(* CODESYS project fablev5.project
   CompiledLibraryCompatibilityVersion: LeadSysStudio V3.5 SP15 Patch 4
   Title: MC500_EtherCAT_axis_motion

Project tree, tasks and I/O mapping:
  Device : MC508, Leadshine Technology Co., Ltd., order no. 508101, version 3.5.15.40
      settings: RetainMode = 0; RetainStartAddr = 20480; RetainEndAddr = 524288; RetainSize = 524288
    application Application
      libraries: Standard, * (System); LS_ModbusMasterlib, 0.0.0.2 (Leadshine Technology Co.Ltd)
      task MainTask (cyclic, interval 4000 µs, priority 1) calls EtherCAT_Master_Leadshine_A.EtherCAT_Task, POU
      program PLC_PRG [LD]: EC_Axis_motion_control
      program POU [ST]
      program POU_1 [ST]
      program POU_3 [ST]
    Resource Usage
    Network Configuration
      LocalBus Config
    Device Diagnose
    LocalBus_Master_Module : LocalBus Master, Leadshine Technology Co., Ltd., version 3.5.15.40
    ModbusCOM_Master_1 : ModbusCOM RS-485 Master, Leadshine Technology Co., Ltd., version 3.5.15.40
        settings: com.Parity = 2; com.FrameIntervTime = 10; com.Baudrate = 115200
      ModbusCOM_Slave : ModbusCOM Slave, Leadshine Technology Co., Ltd., version 3.5.15.40
          settings: ModBusRTU_ErrorCode = 0; Z_Trigger.FuncCode = 6; Z_Trigger.ControlMode = 1; Z_Trigger.ResendCount = 1; Z_Trigger.WriteRegOffSet = 24578; Z_Trigger.IOChannel = 0; Z_Trigger.ChannelName = 'Z_Trigger'; Z_Trigger.ChannelNote = ''; Z_Status.FuncCode = 3; Z_Status.ResendCount = 1; Z_Status.CycleTimes = 50; Z_Status.ReadRegOffSet = 24578; Z_Status.ChannelName = 'Z_Status'; Z_Status.ChannelNote = ''; Z_MotionStat.FuncCode = 3; Z_MotionStat.ResendCount = 1; Z_MotionStat.CycleTimes = 50; Z_MotionStat.ReadRegOffSet = 4099; Z_MotionStat.IOChannel = 2; Z_MotionStat.ChannelName = 'Z_MotionStat'; Z_MotionStat.ChannelNote = ''; Z_Enable.FuncCode = 6; Z_Enable.ControlMode = 1; Z_Enable.ResendCount = 1; Z_Enable.WriteRegOffSet = 15; Z_Enable.IOChannel = 3; Z_Enable.ChannelName = 'Z_Enable'; Z_Enable.ChannelNote = ''; Z_DIStatus.FuncCode = 3; Z_DIStatus.ResendCount = 1; Z_DIStatus.CycleTimes = 200; Z_DIStatus.ReadRegOffSet = 377; Z_DIStatus.IOChannel = 4; Z_DIStatus.ChannelName = 'Z_DIStatus'; Z_DIStatus.ChannelNote = ''; Vendor.SlaveID = 2; Vendor.ChannelNum = 5; Vendor.Timeout = 100
          unmapped channels: ErrorCode, Z_Trigger, Z_Trigger, Z_Trigger, Z_Status, Z_Status, Z_MotionStat, Z_MotionStat, Z_Enable, Z_Enable, Z_Enable, Z_DIStatus, Z_DIStatus
    High_Speed_IO_Module : High Speed IO, Leadshine Technology Co., Ltd., version 3.5.15.40
        unmapped channels: Genral_IO_IN, Genral_IO_Out
    SoftMotion General Axis Pool
    EtherCAT_Master_Leadshine_A : EtherCAT Master SoftMotion, 3S - Smart Software Solutions GmbH, version 3.5.15.30
        settings: NetworkName = 'ecat'; SelectNetworkByName = TRUE
      CS3E_D1008 : CS3E-D1008(COE), Leadshine Technology Co.,Ltd., order no. CS3E-D1008, version Revision=16#00000001
          settings: DC sync0 cycletime = 4000; DC sync1 cycletime = 4000; Number of SDO = 6; Homing method.Index = 16#6098; Homing method.Subindex = 16#00; Homing method.Value = 17; Homing method.Size = 8; Homing method.AbortIfError = FALSE; Homing method.JumpToLine = FALSE; Homing method.Line = 0; Homing method.CompleteAccess = FALSE; Homing velocity (fast).Index = 16#6099; Homing velocity (fast).Subindex = 16#01; Homing velocity (fast).Value = 2000; Homing velocity (fast).Size = 32; Homing velocity (fast).AbortIfError = FALSE; Homing velocity (fast).JumpToLine = FALSE; Homing velocity (fast).Line = 0; Homing velocity (fast).CompleteAccess = FALSE; Homing velocity (slow).Index = 16#6099; Homing velocity (slow).Subindex = 16#02; Homing velocity (slow).Value = 300; Homing velocity (slow).Size = 32; Homing velocity (slow).AbortIfError = FALSE; Homing velocity (slow).JumpToLine = FALSE; Homing velocity (slow).Line = 0; Homing velocity (slow).CompleteAccess = FALSE; Homing acceleration.Index = 16#609A; Homing acceleration.Subindex = 16#00; Homing acceleration.Value = 5000; Homing acceleration.Size = 32; Homing acceleration.AbortIfError = FALSE; Homing acceleration.JumpToLine = FALSE; Homing acceleration.Line = 0; Homing acceleration.CompleteAccess = FALSE; Homing offset.Index = 16#607C; Homing offset.Subindex = 16#00; Homing offset.Value = 0; Homing offset.Size = 32; Homing offset.AbortIfError = FALSE;
            Homing offset.JumpToLine = FALSE; Homing offset.Line = 0; Homing offset.CompleteAccess = FALSE
          unmapped channels: Control Word, Profile Target Position, Touch Probe Function, Last Error Code, Status Word, Modes of Operation display, Position Actual Value, Touch Probe Status, Touch Probe 1 Positive Value, Digital Inputs
        yAxis : Axis, 3S - Smart Software Solutions GmbH, order no. 0, version 4.6.1.0
            settings: wDriveID = 0; dwRatioTechUnitsDenom = 20; eRampType = 3; Number of pulses for one revolution = 4000; The displacement for one revolution of the workbench = 100; Gear ratio molecule = 10; Gear ratio denominator = 10; Home velocity = 100; Home Creep speed = 15.000; Home acceleration = 250; Home position offset = 0; Home velocitySDO = 2000; Home Creep speedSDO = 300; Home position offsetSDO = 0; ScalingIncs = 4000; AdrOffset_8010 = 16; BitOffset_8010 = 0; BitLength_8010 = 16; Address_8010 = '%QW8'; Type_8010 = 'UINT'; AddressPointer_8010 = ADR(%QW8); AdrOffset_8020 = 20; BitOffset_8020 = 0; BitLength_8020 = 32; Address_8020 = '%QD5'; Type_8020 = 'DINT'; AddressPointer_8020 = ADR(%QD5); AdrOffset_8030 = 4294967295; BitOffset_8030 = 0; BitLength_8030 = 0; Address_8030 = ''; Type_8030 = ''; AddressPointer_8030 = 0; AdrOffset_8040 = 4294967295; BitOffset_8040 = 0; BitLength_8040 = 0; Address_8040 = ''; Type_8040 = ''; AddressPointer_8040 = 0; AdrOffset_8050 = 4294967295;
              BitOffset_8050 = 0; BitLength_8050 = 0; Address_8050 = ''; Type_8050 = ''; AddressPointer_8050 = 0; AdrOffset_8060 = 24; BitOffset_8060 = 0; BitLength_8060 = 16; Address_8060 = '%QW12'; Type_8060 = 'UINT'; AddressPointer_8060 = ADR(%QW12); AdrOffset_8070 = 4294967295; BitOffset_8070 = 0; BitLength_8070 = 0; Address_8070 = ''; Type_8070 = ''; AddressPointer_8070 = 0; AdrOffset_8080 = 4294967295; BitOffset_8080 = 0; BitLength_8080 = 0; Address_8080 = ''; Type_8080 = ''; AddressPointer_8080 = 0; AdrOffset_8090 = 4294967295; BitOffset_8090 = 0; BitLength_8090 = 0; Address_8090 = ''; Type_8090 = ''; AddressPointer_8090 = 0; AdrOffset_8510 = 30; BitOffset_8510 = 0; BitLength_8510 = 16; Address_8510 = '%IW15'; Type_8510 = 'UINT'; AddressPointer_8510 = ADR(%IW15); AdrOffset_8520 = 36; BitOffset_8520 = 0; BitLength_8520 = 32; Address_8520 = '%ID9'; Type_8520 = 'DINT';
              AddressPointer_8520 = ADR(%ID9); AdrOffset_8530 = 4294967295; BitOffset_8530 = 0; BitLength_8530 = 0; Address_8530 = ''; Type_8530 = ''; AddressPointer_8530 = 0; AdrOffset_8540 = 4294967295; BitOffset_8540 = 0; BitLength_8540 = 0; Address_8540 = ''; Type_8540 = ''; AddressPointer_8540 = 0; AdrOffset_8550 = 32; BitOffset_8550 = 0; BitLength_8550 = 8; Address_8550 = '%IB32'; Type_8550 = 'SINT'; AddressPointer_8550 = ADR(%IB32); AdrOffset_8560 = 48; BitOffset_8560 = 0; BitLength_8560 = 32; Address_8560 = '%ID12'; Type_8560 = 'UDINT'; AddressPointer_8560 = ADR(%ID12); AdrOffset_8570 = 40; BitOffset_8570 = 0; BitLength_8570 = 16; Address_8570 = '%IW20'; Type_8570 = 'UINT'; AddressPointer_8570 = ADR(%IW20); AdrOffset_8580 = 44; BitOffset_8580 = 0; BitLength_8580 = 32; Address_8580 = '%ID11'; Type_8580 = 'DINT'; AddressPointer_8580 = ADR(%ID11); AdrOffset_8590 = 4294967295; BitOffset_8590 = 0; BitLength_8590 = 0;
              Address_8590 = ''; Type_8590 = ''; AddressPointer_8590 = 0; AdrOffset_8600 = 4294967295; BitOffset_8600 = 0; BitLength_8600 = 0; Address_8600 = ''; Type_8600 = ''; AddressPointer_8600 = 0; AdrOffset_8600 = 4294967295; BitOffset_8600 = 0; BitLength_8600 = 0; Address_8610 = ''; Type_8610 = ''; AddressPointer_8610 = 0; AdrOffset_8620 = 4294967295; BitOffset_8620 = 0; BitLength_8620 = 0; Address_8620 = ''; Type_8620 = ''; AddressPointer_8620 = 0; Home accelerationSDO = 5000
      CS3E_D1008_1 : CS3E-D1008(COE), Leadshine Technology Co.,Ltd., order no. CS3E-D1008, version Revision=16#00000001
          settings: DC sync0 cycletime = 4000; DC sync1 cycletime = 4000; Number of SDO = 6; Homing method.Index = 16#6098; Homing method.Subindex = 16#00; Homing method.Value = 17; Homing method.Size = 8; Homing method.AbortIfError = FALSE; Homing method.JumpToLine = FALSE; Homing method.Line = 0; Homing method.CompleteAccess = False; Homing velocity (fast).Index = 16#6099; Homing velocity (fast).Subindex = 16#01; Homing velocity (fast).Value = 2000; Homing velocity (fast).Size = 32; Homing velocity (fast).AbortIfError = FALSE; Homing velocity (fast).JumpToLine = FALSE; Homing velocity (fast).Line = 0; Homing velocity (fast).CompleteAccess = False; Homing velocity (slow).Index = 16#6099; Homing velocity (slow).Subindex = 16#02; Homing velocity (slow).Value = 300; Homing velocity (slow).Size = 32; Homing velocity (slow).AbortIfError = FALSE; Homing velocity (slow).JumpToLine = FALSE; Homing velocity (slow).Line = 0; Homing velocity (slow).CompleteAccess = False; Homing acceleration.Index = 16#609A; Homing acceleration.Subindex = 16#00; Homing acceleration.Value = 5000; Homing acceleration.Size = 32; Homing acceleration.AbortIfError = FALSE; Homing acceleration.JumpToLine = FALSE; Homing acceleration.Line = 0; Homing acceleration.CompleteAccess = False; Homing offset.Index = 16#607C; Homing offset.Subindex = 16#00; Homing offset.Value = 0; Homing offset.Size = 32; Homing offset.AbortIfError = FALSE;
            Homing offset.JumpToLine = FALSE; Homing offset.Line = 0; Homing offset.CompleteAccess = False
          unmapped channels: Control Word, Profile Target Position, Touch Probe Function, Last Error Code, Status Word, Modes of Operation display, Position Actual Value, Touch Probe Status, Touch Probe 1 Positive Value, Digital Inputs
        XAXIS : Axis, 3S - Smart Software Solutions GmbH, order no. 0, version 4.6.1.0
            settings: dwRatioTechUnitsDenom = 20; Commisioning.smci.Distance = 110; Commisioning.smci.Velocity = 100; Gear ratio molecule = 500; Gear ratio denominator = 500; Home velocity = 100; Home Creep speed = 15; Home acceleration = 250; Home position offset = 0; Home velocitySDO = 2000; Home Creep speedSDO = 300; Home position offsetSDO = 0; ScalingIncs = 4000; InvertDirection = False; AdrOffset_8010 = 4; BitOffset_8010 = 0; BitLength_8010 = 16; Address_8010 = '%QW2'; Type_8010 = 'UINT'; AddressPointer_8010 = ADR(%QW2); AdrOffset_8020 = 8; BitOffset_8020 = 0; BitLength_8020 = 32; Address_8020 = '%QD2'; Type_8020 = 'DINT'; AddressPointer_8020 = ADR(%QD2); AdrOffset_8030 = 4294967295; BitOffset_8030 = 0; BitLength_8030 = 0; Address_8030 = ''; Type_8030 = ''; AddressPointer_8030 = 0; AdrOffset_8040 = 4294967295; BitOffset_8040 = 0; BitLength_8040 = 0; Address_8040 = ''; Type_8040 = ''; AddressPointer_8040 = 0; AdrOffset_8050 = 4294967295; BitOffset_8050 = 0;
              BitLength_8050 = 0; Address_8050 = ''; Type_8050 = ''; AddressPointer_8050 = 0; AdrOffset_8060 = 12; BitOffset_8060 = 0; BitLength_8060 = 16; Address_8060 = '%QW6'; Type_8060 = 'UINT'; AddressPointer_8060 = ADR(%QW6); AdrOffset_8070 = 4294967295; BitOffset_8070 = 0; BitLength_8070 = 0; Address_8070 = ''; Type_8070 = ''; AddressPointer_8070 = 0; AdrOffset_8080 = 4294967295; BitOffset_8080 = 0; BitLength_8080 = 0; Address_8080 = ''; Type_8080 = ''; AddressPointer_8080 = 0; AdrOffset_8090 = 4294967295; BitOffset_8090 = 0; BitLength_8090 = 0; Address_8090 = ''; Type_8090 = ''; AddressPointer_8090 = 0; AdrOffset_8510 = 6; BitOffset_8510 = 0; BitLength_8510 = 16; Address_8510 = '%IW3'; Type_8510 = 'UINT'; AddressPointer_8510 = ADR(%IW3); AdrOffset_8520 = 12; BitOffset_8520 = 0; BitLength_8520 = 32; Address_8520 = '%ID3'; Type_8520 = 'DINT'; AddressPointer_8520 = ADR(%ID3);
              AdrOffset_8530 = 4294967295; BitOffset_8530 = 0; BitLength_8530 = 0; Address_8530 = ''; Type_8530 = ''; AddressPointer_8530 = 0; AdrOffset_8540 = 4294967295; BitOffset_8540 = 0; BitLength_8540 = 0; Address_8540 = ''; Type_8540 = ''; AddressPointer_8540 = 0; AdrOffset_8550 = 8; BitOffset_8550 = 0; BitLength_8550 = 8; Address_8550 = '%IB8'; Type_8550 = 'SINT'; AddressPointer_8550 = ADR(%IB8); AdrOffset_8560 = 24; BitOffset_8560 = 0; BitLength_8560 = 32; Address_8560 = '%ID6'; Type_8560 = 'UDINT'; AddressPointer_8560 = ADR(%ID6); AdrOffset_8570 = 16; BitOffset_8570 = 0; BitLength_8570 = 16; Address_8570 = '%IW8'; Type_8570 = 'UINT'; AddressPointer_8570 = ADR(%IW8); AdrOffset_8580 = 20; BitOffset_8580 = 0; BitLength_8580 = 32; Address_8580 = '%ID5'; Type_8580 = 'DINT'; AddressPointer_8580 = ADR(%ID5); AdrOffset_8590 = 4294967295; BitOffset_8590 = 0; BitLength_8590 = 0; Address_8590 = '';
              Type_8590 = ''; AddressPointer_8590 = 0; AdrOffset_8600 = 4294967295; BitOffset_8600 = 0; BitLength_8600 = 0; Address_8600 = ''; Type_8600 = ''; AddressPointer_8600 = 0; AdrOffset_8600 = 4294967295; BitOffset_8600 = 0; BitLength_8600 = 0; Address_8610 = ''; Type_8610 = ''; AddressPointer_8610 = 0; AdrOffset_8620 = 4294967295; BitOffset_8620 = 0; BitLength_8620 = 0; Address_8620 = ''; Type_8620 = ''; AddressPointer_8620 = 0; Home accelerationSDO = 5000
*)

// Device/Application/POU
PROGRAM POU
VAR
    // ===== X/Y ETHERCAT AXES =====
    MC_Power_1 : MC_Power;    MC_Power_2 : MC_Power;
    MC_Home_1  : MC_Home;     MC_Home_2  : MC_Home;
    MC_Reset_1 : MC_Reset;    MC_Reset_2 : MC_Reset;
    MC_Stop_1  : MC_Stop;     MC_Stop_2  : MC_Stop;

    LS_MoveXY : LS_2AxisLine;
    TargetXY  : ARRAY[0..1] OF LREAL := [0.0, 0.0];

    // ===== Z AXIS MODBUS (CS2RS-D1008) — trigger-mode channels =====
    Z_Trigger    AT %QW13   : WORD := 0;
    Z_Status     AT %IW28   : WORD := 0;   // readback of 0x6002
    Z_MotionStat AT %IW30   : WORD := 0;   // 0x1003
    Z_Enable     AT %QW15   : WORD := 1;   // NOTE: shifted to QW15
    Z_DIStatus   AT %IW32   : WORD := 0;
    Z_Trigger_Send AT %QX28.0 : BOOL := FALSE;  // trigger control bit
    Z_Enable_Send  AT %QX32.0 : BOOL := FALSE;  // trigger control bit
    Z_Trig_Done    AT %IX54.0 : BOOL;           // processing complete state
    ModbusErr      AT %IW26   : WORD;

    // ===== Z COMMAND SENDER (closed loop) =====
    z_send_step    : INT  := 0;
    z_cmd_request  : BOOL := FALSE;
    z_cmd_value    : WORD := 0;
    z_stop_request : BOOL := FALSE;
    z_retry_count  : INT  := 0;
    Z_MAX_RETRY    : INT  := 3;
    z_ack_timer    : TON;
    Z_ACK_TIMEOUT  : TIME := T#250MS;
    z_verify_timer : TON;
    Z_VERIFY_T     : TIME := T#400MS;
    z_cmd_fault    : BOOL := FALSE;
    z_enable_sent  : BOOL := FALSE;
    z_en_pulse     : TON;
    Z_EN_PULSE_T   : TIME := T#100MS;

    // ===== Z MOVE SUPERVISOR (shared completion handler) =====
    z_next_state   : INT  := 0;      // where to go after Z confirms arrival
    z_issue_state  : INT  := 0;      // state that issued the Z command
    z_saw_running  : BOOL := FALSE;

    // ===== END EFFECTOR =====
    end_effector AT %QX1.4 : BOOL := FALSE;

    // ===== BUTTONS =====
    btn_a AT %IX0.0 : BOOL := FALSE;
    btn_b AT %IX0.1 : BOOL := FALSE;
    sw_a : BOOL := FALSE;   sw_b : BOOL := FALSE;
    rt_a : R_TRIG;          rt_b : R_TRIG;
    pending_start   : BOOL := FALSE;
    pending_pause   : BOOL := FALSE;
    pending_resume  : BOOL := FALSE;
    pending_restart : BOOL := FALSE;

    // ===== TEST LOOP MODE =====
    // TRUE  = endless cycling with a dwell between cycles (testing)
    // FALSE = stop in state 91 and wait for operator (production)
    TEST_LOOP_MODE : BOOL := TRUE;
    loop_dwell     : TON;
    LOOP_DWELL_T   : TIME := T#3S;
    cycle_count    : UDINT := 0;

    // ===== TIMERS =====
    grip_timer   : TON;
    GRIP_TIME    : TIME := T#500MS;
    RELEASE_TIME : TIME := T#500MS;
    stop_release_timer  : TON;
    STOP_RELEASE_TIME   : TIME := T#200MS;
    stop_release_done   : BOOL := FALSE;
    home_teardown_timer : TON;
    HOME_TEARDOWN_TIME  : TIME := T#50MS;
    home_teardown_done  : BOOL := FALSE;

  // ===== TRAY CONFIGURATION =====
    PICK_BASE_X     : LREAL := 145.0  ;
    PICK_BASE_Y     : LREAL := 45.0;
    PICK_SPACING_X  : LREAL := 80.0;          // 30 mm pick pitch
    PICK_SPACING_Y  : LREAL := 80.0;          // 30 mm pick pitch
    PLACE_BASE_X    : LREAL := 740.0;        // top-centre slot X when griddle is at drop-zone
    PLACE_BASE_Y    : LREAL := 116.0;          // top-centre slot Y when griddle is at drop-zone

    // Griddle slot offsets — diamond layout (1-top, 2×2-mid, 1-bottom), 380 mm span
    // Calibrate PLACE_OFFSET_X col half-pitch (currently ±55 mm) and Y rows after physical run.
    // Index:          0      1       2      3       4      5
    PLACE_OFFSET_X  : ARRAY[0..5] OF LREAL := [ 0.0, 70.0,  -70.0, 70.0,  -70.0,  0.0];
    PLACE_OFFSET_Y  : ARRAY[0..5] OF LREAL := [ 0.0, 66.0, 66.0, 143.0, 143.0, 210.0];

    TRAY_COLS           : INT := 6;           // pick grid — 6 columns
    TRAY_ROWS           : INT := 4;           // pick grid — 4 rows
    TOTAL_PATTIES       : INT := 24;          // 4 × 6
    PATTIES_PER_GRIDDLE : INT := 6;           // slots per griddle
    GRIDDLE_COUNT       : INT := 4;           // griddles on rotating tray
    patty_index   : INT := 0;
    current_col   : INT := 0;   current_row   : INT := 0;
    griddle_index : INT := 0;                 // which griddle (0-3)
    slot_index    : INT := 0;                 // slot within current griddle (0-5)
    pick_x  : LREAL := 0.0;   pick_y  : LREAL := 0.0;
    place_x : LREAL := 0.0;   place_y : LREAL := 0.0;

    // ===== GRIDDLE ROTATION (timed dwell — swap for I/O handshake when drive fitted) =====
    griddle_dwell   : TON;
    GRIDDLE_DWELL_T : TIME := T#5S;           // set to actual rotation time
    // ===== STATE MACHINE =====
    state          : INT := 0;
    saved_state    : INT := 0;
    saved_TargetX  : LREAL := 0.0;
    saved_TargetY  : LREAL := 0.0;
    drive_enable   : BOOL := TRUE;
    paused         : BOOL := FALSE;
    cycle_complete : BOOL := FALSE;
    cycle_active   : BOOL := FALSE;
    stop_method    : INT := 0;

    // ===== Z STATUS DECODE =====
    z_status_val  : WORD := 0;
    z_motion_stat : WORD := 0;
    z_homing_done : BOOL := FALSE;
    z_is_running  : BOOL := FALSE;
    z_path_done   : BOOL := FALSE;
    z_has_fault   : BOOL := FALSE;
    z_is_enabled  : BOOL := FALSE;

    // ===== TIMING (scan counts @ 4 ms task) =====
    z_wait_count   : INT := 0;
    Z_MIN_WAIT     : INT := 75;     // 300 ms: cmd out + fresh status read
    Z_IDLE_CONFIRM : INT := 50;     // 200 ms stable idle
    Z_HOME_WAIT    : INT := 7500;   // 30 s homing timeout
    Z_MOVE_TIMEOUT : INT := 2500;   // 10 s per Z move, then FAULT
    xy_home_timer  : INT := 0;
    XY_HOME_WAIT   : INT := 7500;

    QUICK_STOP_DECEL : LREAL := 3000.0;
    hmi_start   : BOOL := FALSE;
    hmi_restart : BOOL := FALSE;
END_VAR

// =====================================================================
// EDGE DETECTION + BUTTONS
// =====================================================================
rt_a(CLK := btn_a OR sw_a OR hmi_start);
rt_b(CLK := btn_b OR sw_b OR hmi_restart);
sw_a := FALSE;  sw_b := FALSE;
hmi_start := FALSE;  hmi_restart := FALSE;

IF rt_a.Q THEN
    IF NOT cycle_active AND NOT paused THEN
        pending_start := TRUE;
    ELSIF cycle_active AND NOT paused THEN
        pending_pause := TRUE;
    ELSIF paused THEN
        pending_resume := TRUE;
    END_IF
END_IF
IF rt_b.Q THEN
    pending_restart := TRUE;
END_IF

// =====================================================================
// PAUSE TRIGGER
// =====================================================================
IF (pending_pause OR pending_restart) AND cycle_active AND state <> 200 THEN
    saved_state   := state;
    saved_TargetX := TargetXY[0];
    saved_TargetY := TargetXY[1];

    IF LS_MoveXY.Busy THEN
        stop_method := 1;
        LS_MoveXY.Exec := FALSE;
    ELSIF state = 1 THEN
        stop_method := 2;
        MC_Home_1(Axis := yAxis, Execute := FALSE, Position := 0);
        MC_Home_2(Axis := XAXIS, Execute := FALSE, Position := 0);
    ELSE
        stop_method := 3;
    END_IF

    z_stop_request := TRUE;            // sender delivers 0x0040 with priority
    griddle_dwell(IN := FALSE);    // ← ADD — abort in-flight rotation dwell

    paused        := TRUE;
    cycle_active  := FALSE;
    pending_pause := FALSE;
    stop_release_done := FALSE;
    stop_release_timer(IN := FALSE);
    home_teardown_done := FALSE;
    home_teardown_timer(IN := FALSE);
    state := 200;
END_IF

// =====================================================================
// SENDER FAULT → ERROR STATE (not while paused)
// =====================================================================
IF z_cmd_fault AND state <> 200 THEN
    z_cmd_fault := FALSE;
    state := 199;
END_IF

// =====================================================================
// POWER + Z DECODE
// =====================================================================
MC_Power_1(Axis := yAxis, Enable := drive_enable, bRegulatorOn := TRUE, bDriveStart := TRUE);
MC_Power_2(Axis := XAXIS, Enable := drive_enable, bRegulatorOn := TRUE, bDriveStart := TRUE);

z_status_val  := Z_Status;
z_motion_stat := Z_MotionStat;
z_has_fault   := (z_motion_stat AND 16#0001) <> 0;
z_is_enabled  := (z_motion_stat AND 16#0002) <> 0;
z_is_running  := (z_motion_stat AND 16#0004) <> 0;
z_path_done   := (z_motion_stat AND 16#0020) <> 0;
z_homing_done := (z_motion_stat AND 16#0040) <> 0;

// =====================================================================
// MAIN STATE MACHINE
// =====================================================================
CASE state OF

// ---------- STATE 0: IDLE / TEARDOWN ----------
0:
    cycle_complete := FALSE;
    cycle_active   := FALSE;
    paused         := FALSE;
    end_effector   := FALSE;
    stop_method    := 0;
    z_wait_count   := 0;
    xy_home_timer  := 0;
    griddle_index  := 0;        // reset griddle counter each cycle
    slot_index     := 0;        // reset slot counter
    griddle_dwell(IN := FALSE); // reset rotation dwell timer

    IF NOT z_enable_sent THEN   // one-shot Z enable after PLC start
        Z_Enable := 1;
        Z_Enable_Send := TRUE;
        z_en_pulse(IN := TRUE, PT := Z_EN_PULSE_T);
        IF z_en_pulse.Q THEN
            Z_Enable_Send := FALSE;
            z_en_pulse(IN := FALSE);
            z_enable_sent := TRUE;
        END_IF
    END_IF

    LS_MoveXY.Exec := FALSE;
    MC_Home_1(Axis := yAxis, Execute := FALSE, Position := 0);
    MC_Home_2(Axis := XAXIS, Execute := FALSE, Position := 0);
    MC_Stop_1(Axis := yAxis, Execute := FALSE, Deceleration := QUICK_STOP_DECEL);
    MC_Stop_2(Axis := XAXIS, Execute := FALSE, Deceleration := QUICK_STOP_DECEL);

    IF pending_start OR pending_restart THEN
        pending_start   := FALSE;
        pending_restart := FALSE;
        IF MC_Power_1.Status AND MC_Power_2.Status THEN
            patty_index := 0;
            cycle_active := TRUE;
            state := 1;
        END_IF
    END_IF
	
// ---------- STATE 1: HOME X AND Y ----------
1:
    MC_Home_1(Axis := yAxis, Execute := TRUE, Position := 0);
    MC_Home_2(Axis := XAXIS, Execute := TRUE, Position := 0);
    xy_home_timer := xy_home_timer + 1;

    IF (MC_Home_1.Done AND MC_Home_2.Done) OR (xy_home_timer >= XY_HOME_WAIT) THEN
        MC_Home_1(Axis := yAxis, Execute := FALSE, Position := 0);
        MC_Home_2(Axis := XAXIS, Execute := FALSE, Position := 0);
        xy_home_timer := 0;
        z_wait_count := 0;
        state := 2;
    END_IF

// ---------- STATE 2: Z — WAIT IDLE, COMMAND HOMING ----------
// Tolerates power-up auto-homing still in progress (Pr8.00 bit2)
2:
    IF z_is_running OR z_cmd_request THEN
        z_wait_count := 0;
    ELSE
        z_wait_count := z_wait_count + 1;
    END_IF
    IF z_wait_count >= Z_IDLE_CONFIRM THEN
        z_cmd_value := 16#0020;        // write 0x0020 to 0x6002 = home
        z_cmd_request := TRUE;
        z_wait_count := 0;
        state := 3;
    END_IF

// ---------- STATE 3: Z — WAIT HOMING START ----------
3:
    z_wait_count := z_wait_count + 1;
    IF z_wait_count < Z_MIN_WAIT OR z_cmd_request THEN ;
    ELSIF z_is_running THEN
        z_wait_count := 0;
        state := 4;
    ELSIF z_homing_done THEN           // very short home
        state := 10;
    ELSIF z_wait_count >= Z_HOME_WAIT THEN
        state := 199;
    END_IF

// ---------- STATE 4: Z — WAIT HOMING COMPLETE ----------
4:
    z_wait_count := z_wait_count + 1;
    IF NOT z_is_running AND z_homing_done THEN
        state := 10;
    ELSIF z_wait_count >= Z_HOME_WAIT THEN
        state := 199;
    END_IF

// ---------- STATE 10: GRID CALCULATION ----------
10:
    // ── PICK: 4-col × 6-row rectangular grid, 30 mm pitch ──
    current_row := patty_index / TRAY_COLS;          // 0 … 5
    current_col := patty_index MOD TRAY_COLS;        // 0 … 3
    pick_x := PICK_BASE_X + INT_TO_LREAL(current_col) * PICK_SPACING_X;
    pick_y := PICK_BASE_Y + INT_TO_LREAL(current_row) * PICK_SPACING_Y;

    // ── PLACE: diamond-layout griddle slots via offset table ──
    griddle_index := patty_index / PATTIES_PER_GRIDDLE;   // 0 … 3
    slot_index    := patty_index MOD PATTIES_PER_GRIDDLE;  // 0 … 5
    place_x := PLACE_BASE_X + PLACE_OFFSET_X[slot_index];
    place_y := PLACE_BASE_Y + PLACE_OFFSET_Y[slot_index];

    // Rotate to next griddle only at slot 0 of each new griddle (skip at patty 0)
    IF (slot_index = 0) AND (patty_index > 0) THEN
        state := 11;        // dwell for griddle rotation, then pick
    ELSE
        state := 20;
    END_IF

// ---------- STATE 11: GRIDDLE ROTATION DWELL ----------
// Waits GRIDDLE_DWELL_T for the tray to rotate the next griddle into position.
// TODO: replace timer with I/O handshake when the rotation drive is commissioned.
11:
    griddle_dwell(IN := TRUE, PT := GRIDDLE_DWELL_T);
    IF griddle_dwell.Q THEN
        griddle_dwell(IN := FALSE);
        state := 20;
    END_IF
	
// ---------- STATE 20: XY → PICK ----------
20:
    TargetXY[0] := pick_x;
    TargetXY[1] := pick_y;
    LS_MoveXY.Exec := TRUE;
    IF LS_MoveXY.Done THEN
        LS_MoveXY.Exec := FALSE;
        state := 30;
    ELSIF LS_MoveXY.Error THEN
        LS_MoveXY.Exec := FALSE;
        state := 199;
    END_IF

// ---------- Z COMMAND ISSUE STATES (all use shared 100/101) ----------
30: // Z DOWN to pick
    z_cmd_value := 16#0012;  z_next_state := 33;  z_issue_state := 30;
    z_cmd_request := TRUE;   state := 100;

40: // Z UP with patty
    z_cmd_value := 16#0011;  z_next_state := 50;  z_issue_state := 40;
    z_cmd_request := TRUE;   state := 100;

60: // Z DOWN to place
    z_cmd_value := 16#0012;  z_next_state := 63;  z_issue_state := 60;
    z_cmd_request := TRUE;   state := 100;

70: // Z UP after place
    z_cmd_value := 16#0011;  z_next_state := 80;  z_issue_state := 70;
    z_cmd_request := TRUE;   state := 100;

// ---------- STATE 33: GRIP — only reached after CONFIRMED Z arrival ----------
33:
    end_effector := TRUE;
    grip_timer(IN := TRUE, PT := GRIP_TIME);
    IF grip_timer.Q THEN
        grip_timer(IN := FALSE);
        state := 40;
    END_IF

// ---------- STATE 50: XY → PLACE ----------
50:
    TargetXY[0] := place_x;
    TargetXY[1] := place_y;
    LS_MoveXY.Exec := TRUE;
    IF LS_MoveXY.Done THEN
        LS_MoveXY.Exec := FALSE;
        state := 60;
    ELSIF LS_MoveXY.Error THEN
        LS_MoveXY.Exec := FALSE;
        state := 199;
    END_IF

// ---------- STATE 63: RELEASE — only after CONFIRMED Z arrival ----------
63:
    end_effector := FALSE;
    grip_timer(IN := TRUE, PT := RELEASE_TIME);
    IF grip_timer.Q THEN
        grip_timer(IN := FALSE);
        state := 70;
    END_IF

// ---------- STATE 80: NEXT OR DONE ----------
80:
    patty_index := patty_index + 1;
    IF patty_index >= TOTAL_PATTIES THEN
        state := 90;
    ELSE
        state := 10;
    END_IF

// ---------- STATE 90: PARK ----------
90:
    TargetXY[0] := 50.0;
    TargetXY[1] := 50.0;
    LS_MoveXY.Exec := TRUE;
    IF LS_MoveXY.Done OR LS_MoveXY.Error THEN
        LS_MoveXY.Exec := FALSE;
        cycle_complete := TRUE;
        cycle_active   := FALSE;
        cycle_count := cycle_count + 1;
        state := 91;
    END_IF

// ---------- STATE 91: WAIT / TEST LOOP ----------
91:
    IF TEST_LOOP_MODE THEN
        // ===== TEST ONLY: auto-restart after dwell. Re-homes all axes
        // every cycle, so it also stress-tests the Z homing handshake.
        loop_dwell(IN := TRUE, PT := LOOP_DWELL_T);
        IF loop_dwell.Q THEN
            loop_dwell(IN := FALSE);
            cycle_complete := FALSE;
            patty_index := 0;
            cycle_active := TRUE;
            z_wait_count := 0;
            xy_home_timer := 0;
            state := 1;
        END_IF
        // ===== END TEST ONLY
    END_IF

    IF pending_start OR pending_restart THEN
        pending_start   := FALSE;
        pending_restart := FALSE;
        loop_dwell(IN := FALSE);
        cycle_complete := FALSE;
        patty_index := 0;
        cycle_active := TRUE;
        z_wait_count := 0;
        xy_home_timer := 0;
        state := 1;                    // full re-home incl. Z
    END_IF

// =====================================================================
// STATE 100: Z — WAIT SENDER CONFIRMS COMMAND ACCEPTED
// =====================================================================
100:
    IF NOT z_cmd_request AND z_send_step = 0 THEN
        z_wait_count  := 0;
        z_saw_running := z_is_running;
        state := 101;
    END_IF

// =====================================================================
// STATE 101: Z — WAIT CONFIRMED ARRIVAL (strict — no blind fallback)
// Grip/release states are ONLY reachable through here.
// =====================================================================
101:
    z_wait_count := z_wait_count + 1;
    IF z_is_running THEN
        z_saw_running := TRUE;
    END_IF

    IF z_saw_running AND NOT z_is_running
       AND (z_path_done OR z_status_val = 16#0000 OR z_status_val = 16#0200) THEN
        state := z_next_state;                       // motion ran + finished
    ELSIF NOT z_saw_running AND z_status_val = 16#0000
          AND z_wait_count >= Z_MIN_WAIT THEN
        state := z_next_state;                       // zero-distance abs move
    ELSIF z_wait_count >= Z_MOVE_TIMEOUT THEN
        state := 199;                                // never confirmed → FAULT
    END_IF

// ---------- STATE 199: ERROR ----------
199:
    LS_MoveXY.Exec := FALSE;
    end_effector := FALSE;
	griddle_dwell(IN := FALSE);    // ← ADD
    IF pending_restart THEN
        pending_restart := FALSE;
        state := 0;
    END_IF

// ---------- STATE 200: PAUSED ----------
200:
    LS_MoveXY.Exec := FALSE;

    IF stop_method = 1 THEN
        home_teardown_done := TRUE;
    ELSIF stop_method = 2 THEN
        MC_Home_1(Axis := yAxis, Execute := FALSE, Position := 0);
        MC_Home_2(Axis := XAXIS, Execute := FALSE, Position := 0);
        home_teardown_timer(IN := TRUE, PT := HOME_TEARDOWN_TIME);
        IF home_teardown_timer.Q AND NOT home_teardown_done THEN
            MC_Stop_1(Axis := yAxis, Execute := TRUE, Deceleration := QUICK_STOP_DECEL);
            MC_Stop_2(Axis := XAXIS, Execute := TRUE, Deceleration := QUICK_STOP_DECEL);
            home_teardown_done := TRUE;
        END_IF
        IF home_teardown_done AND MC_Stop_1.Done AND MC_Stop_2.Done THEN
            MC_Stop_1(Axis := yAxis, Execute := FALSE, Deceleration := QUICK_STOP_DECEL);
            MC_Stop_2(Axis := XAXIS, Execute := FALSE, Deceleration := QUICK_STOP_DECEL);
        END_IF
    ELSIF stop_method = 3 THEN
        MC_Home_1(Axis := yAxis, Execute := FALSE, Position := 0);
        MC_Home_2(Axis := XAXIS, Execute := FALSE, Position := 0);
        MC_Stop_1(Axis := yAxis, Execute := FALSE, Deceleration := QUICK_STOP_DECEL);
        MC_Stop_2(Axis := XAXIS, Execute := FALSE, Deceleration := QUICK_STOP_DECEL);
        home_teardown_done := TRUE;
    END_IF

    IF home_teardown_done THEN
        stop_release_timer(IN := TRUE, PT := STOP_RELEASE_TIME);
        IF stop_release_timer.Q THEN
            stop_release_done := TRUE;
        END_IF
    END_IF

    IF stop_release_done THEN
        IF pending_restart THEN
            pending_restart := FALSE;  pending_pause := FALSE;
            pending_resume  := FALSE;  paused := FALSE;
            stop_method := 0;          drive_enable := TRUE;
            end_effector := FALSE;     cycle_active := FALSE;
            stop_release_timer(IN := FALSE);  stop_release_done := FALSE;
            home_teardown_timer(IN := FALSE); home_teardown_done := FALSE;
            state := 0;
        ELSIF pending_resume THEN
            pending_resume := FALSE;   paused := FALSE;
            stop_method := 0;          cycle_active := TRUE;
            TargetXY[0] := saved_TargetX;
            TargetXY[1] := saved_TargetY;
            stop_release_timer(IN := FALSE);  stop_release_done := FALSE;
            home_teardown_timer(IN := FALSE); home_teardown_done := FALSE;
            IF saved_state <= 4 THEN
                state := 1;                  // paused during homing → re-home
            ELSIF saved_state >= 100 THEN
                state := z_issue_state;      // re-issue interrupted Z move
            ELSE
                state := saved_state;
            END_IF
        END_IF
    END_IF

END_CASE

// =====================================================================
// Z COMMAND SENDER — closed loop with retry (absolute paths = retry-safe)
// =====================================================================
IF z_stop_request AND z_send_step = 0 AND NOT z_cmd_request THEN
    z_cmd_value := 16#0040;
    z_cmd_request := TRUE;
    z_stop_request := FALSE;
END_IF

CASE z_send_step OF
0:
    IF z_cmd_request THEN
        z_retry_count := 0;
        z_send_step := 1;
    END_IF
1:  // transmit, wait channel ack
    Z_Trigger := z_cmd_value;
    Z_Trigger_Send := TRUE;
    z_ack_timer(IN := TRUE, PT := Z_ACK_TIMEOUT);
    IF Z_Trig_Done THEN
        Z_Trigger_Send := FALSE;
        z_ack_timer(IN := FALSE);
        z_verify_timer(IN := FALSE);
        z_send_step := 2;
    ELSIF z_ack_timer.Q THEN
        Z_Trigger_Send := FALSE;
        z_ack_timer(IN := FALSE);
        z_send_step := 3;
    END_IF
2:  // verify drive acted
    z_verify_timer(IN := TRUE, PT := Z_VERIFY_T);
    IF (z_status_val = z_cmd_value)
       OR ((z_status_val AND 16#0100) <> 0)
       OR (z_status_val = 16#0200)
       OR (z_status_val = 16#0000 AND z_cmd_value <> 16#0020)  // instant abs move
       OR z_is_running
       OR (z_cmd_value = 16#0040)
    THEN
        z_verify_timer(IN := FALSE);
        z_cmd_request := FALSE;
        z_send_step := 0;
    ELSIF z_verify_timer.Q THEN
        z_verify_timer(IN := FALSE);
        z_send_step := 3;
    END_IF
3:  // retry gap (creates fresh rising edge)
    z_retry_count := z_retry_count + 1;
    IF z_retry_count > Z_MAX_RETRY THEN
        z_cmd_request := FALSE;
        z_cmd_fault := TRUE;
        z_send_step := 0;
    ELSE
        z_send_step := 1;
    END_IF
END_CASE

// =====================================================================
// XY INTERPOLATION
// =====================================================================
LS_MoveXY(
    Axis0 := XAXIS, Axis1 := yAxis,
    Halt := FALSE, Stop := paused,
    IpoCycle := 4000, PosMode := 0,
    EndPos := TargetXY, VelocityMode := 4,
    Velocity := 1000, Acceleration := 3000,
    Deceleration := 3000, Jerk := 9000
);

END_PROGRAM

// Device/Application/PLC_PRG
PROGRAM PLC_PRG

VAR
	MC_Power_1: MC_Power;
	MC_Jog_1: MC_JOG;
	ec_enable: BOOL;
	drive_enable: BOOL;
	drive_ready: BOOL;
	homing_ex: BOOL;
	slow: LREAL;
	fast: LREAL;
	acc: LREAL;
	dec: LREAL;
	homing_en: BOOL;
	MC_Power_2: MC_Power;
	MC_Home_1: MC_Home;
	MC_MoveAbsolute_1: MC_MoveAbsolute;
	MC_Reset_1: MC_Reset;
	MC_Home_2: MC_Home;
	MC_MoveAbsolute_2: MC_MoveAbsolute;
	MC_Reset_2: MC_Reset;
	MC_MoveAbsolute_3: MC_MoveAbsolute;
	MC_MoveAbsolute_4: MC_MoveAbsolute;
	MC_MoveAbsolute_5: MC_MoveAbsolute;
	MC_MoveAbsolute_6: MC_MoveAbsolute;
	MC_MoveAbsolute_7: MC_MoveAbsolute;
	MC_MoveAbsolute_8: MC_MoveAbsolute;
	MC_MoveAbsolute_9: MC_MoveAbsolute;
	MC_MoveAbsolute_10: MC_MoveAbsolute;
	LS_2AxisLine_0: LS_2AxisLine;
	EndPosition : ARRAY[0..1] OF LREAL := [-6.0, 1.5];
	EndPosition1 : ARRAY[0..1] OF LREAL := [-1.0, 0.5];
	LS_2AxisLine_1: LS_2AxisLine;
END_VAR

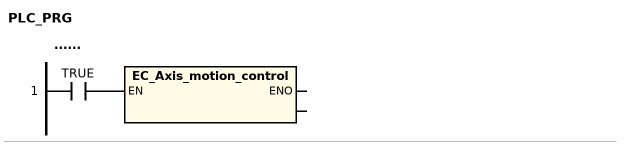
// NETWORK 1: ......
EC_Axis_motion_control();

ACTION EC_Axis_motion_control:
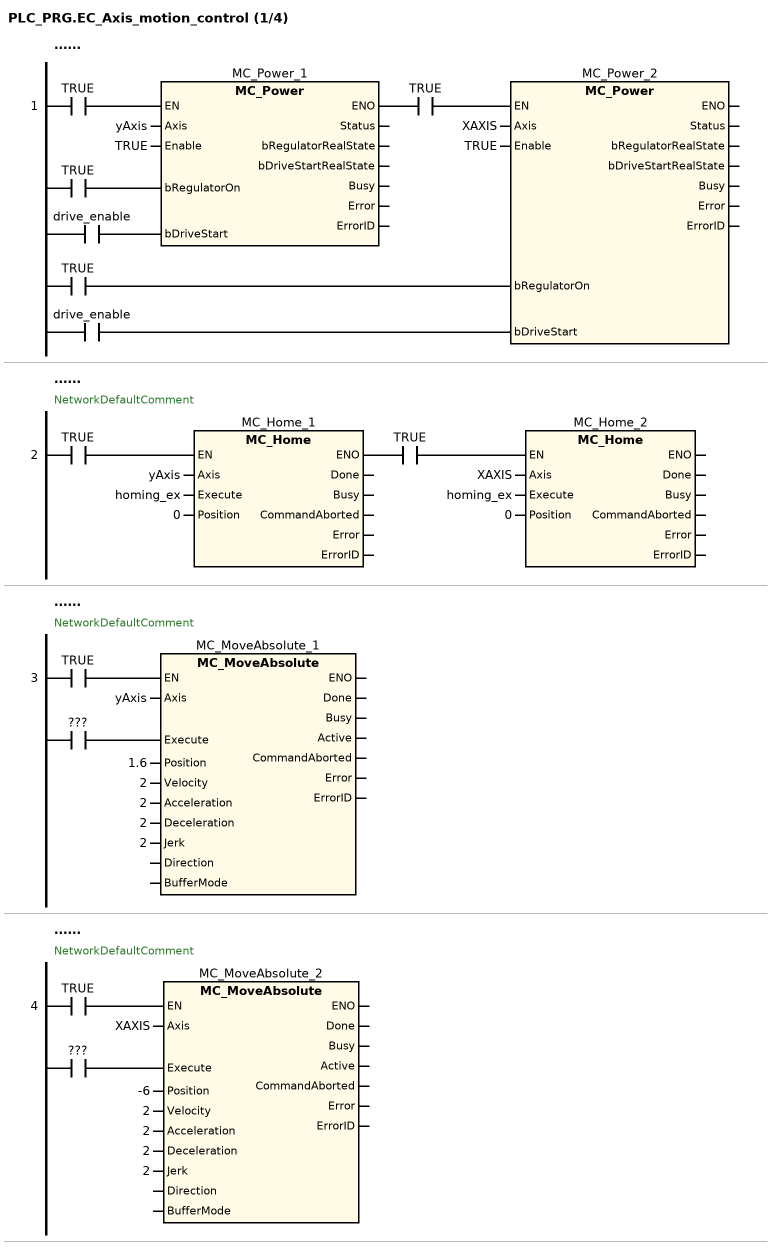
// NETWORK 1: ......
MC_Power_1(Axis := yAxis, Enable := TRUE, bRegulatorOn := TRUE, bDriveStart := drive_enable); // MC_Power
IF TRUE AND TRUE THEN
    MC_Power_2(Axis := XAXIS, Enable := TRUE, bRegulatorOn := TRUE, bDriveStart := drive_enable); // MC_Power
END_IF

// NETWORK 2: ......
// NetworkDefaultComment
MC_Home_1(Axis := yAxis, Execute := homing_ex, Position := 0); // MC_Home
IF TRUE AND TRUE THEN
    MC_Home_2(Axis := XAXIS, Execute := homing_ex, Position := 0); // MC_Home
END_IF

// NETWORK 3: ......
// NetworkDefaultComment
MC_MoveAbsolute_1(
    Axis := yAxis,
    Position := 1.6,
    Velocity := 2,
    Acceleration := 2,
    Deceleration := 2,
    Jerk := 2); // MC_MoveAbsolute

// NETWORK 4: ......
// NetworkDefaultComment
MC_MoveAbsolute_2(
    Axis := XAXIS,
    Position := -6,
    Velocity := 2,
    Acceleration := 2,
    Deceleration := 2,
    Jerk := 2); // MC_MoveAbsolute

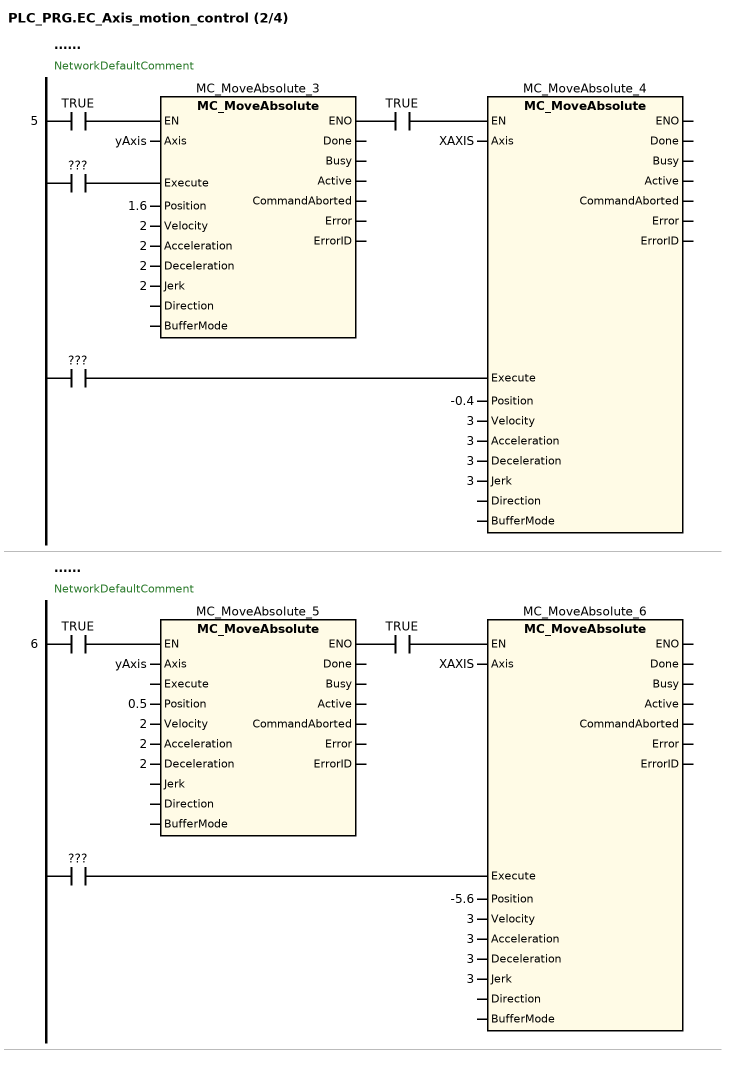
// NETWORK 5: ......
// NetworkDefaultComment
MC_MoveAbsolute_3(
    Axis := yAxis,
    Position := 1.6,
    Velocity := 2,
    Acceleration := 2,
    Deceleration := 2,
    Jerk := 2); // MC_MoveAbsolute
IF TRUE AND TRUE THEN
    MC_MoveAbsolute_4(
        Axis := XAXIS,
        Position := -0.4,
        Velocity := 3,
        Acceleration := 3,
        Deceleration := 3,
        Jerk := 3); // MC_MoveAbsolute
END_IF

// NETWORK 6: ......
// NetworkDefaultComment
MC_MoveAbsolute_5(Axis := yAxis, Position := 0.5, Velocity := 2, Acceleration := 2, Deceleration := 2); // MC_MoveAbsolute
IF TRUE AND TRUE THEN
    MC_MoveAbsolute_6(
        Axis := XAXIS,
        Position := -5.6,
        Velocity := 3,
        Acceleration := 3,
        Deceleration := 3,
        Jerk := 3); // MC_MoveAbsolute
END_IF

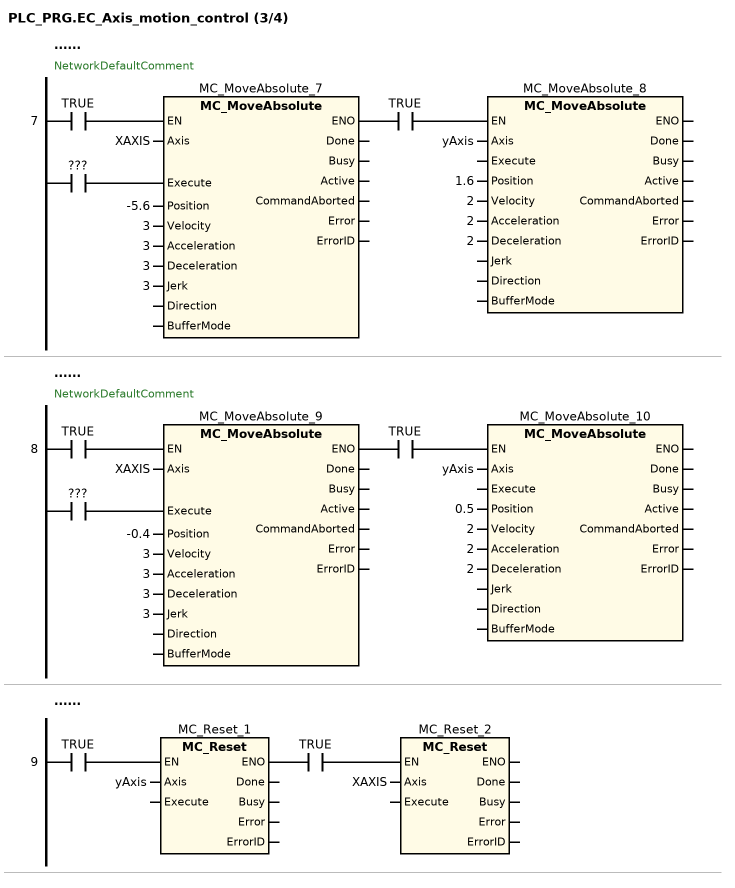
// NETWORK 7: ......
// NetworkDefaultComment
MC_MoveAbsolute_7(
    Axis := XAXIS,
    Position := -5.6,
    Velocity := 3,
    Acceleration := 3,
    Deceleration := 3,
    Jerk := 3); // MC_MoveAbsolute
IF TRUE AND TRUE THEN
    MC_MoveAbsolute_8(Axis := yAxis, Position := 1.6, Velocity := 2, Acceleration := 2, Deceleration := 2); // MC_MoveAbsolute
END_IF

// NETWORK 8: ......
// NetworkDefaultComment
MC_MoveAbsolute_9(
    Axis := XAXIS,
    Position := -0.4,
    Velocity := 3,
    Acceleration := 3,
    Deceleration := 3,
    Jerk := 3); // MC_MoveAbsolute
IF TRUE AND TRUE THEN
    MC_MoveAbsolute_10(Axis := yAxis, Position := 0.5, Velocity := 2, Acceleration := 2, Deceleration := 2); // MC_MoveAbsolute
END_IF

// NETWORK 9: ......
MC_Reset_1(Axis := yAxis); // MC_Reset
IF TRUE AND TRUE THEN
    MC_Reset_2(Axis := XAXIS); // MC_Reset
END_IF

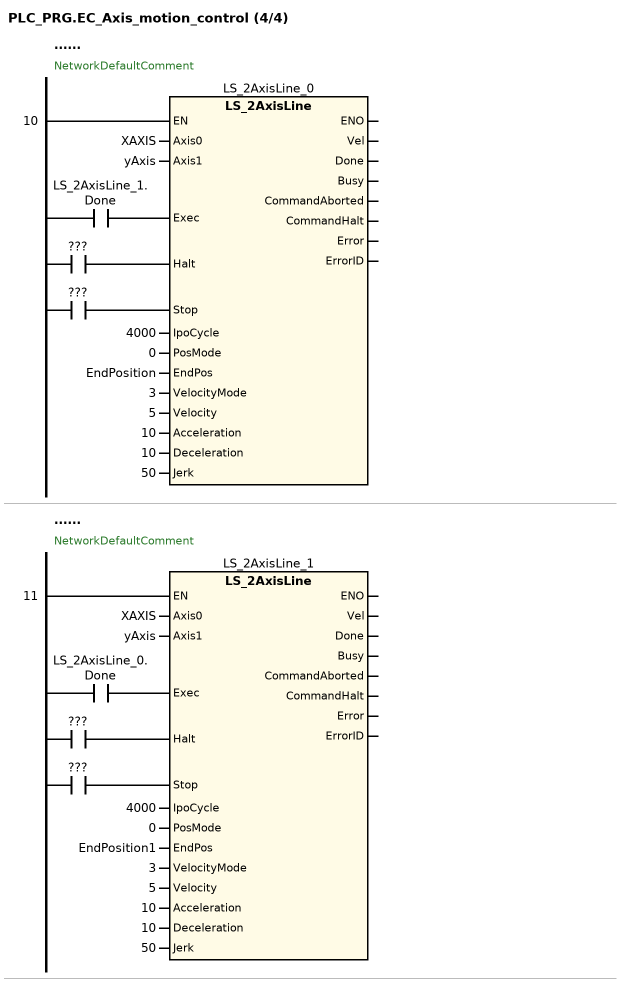
// NETWORK 10: ......
// NetworkDefaultComment
LS_2AxisLine_0(
    Axis0 := XAXIS,
    Axis1 := yAxis,
    Exec := LS_2AxisLine_1.Done,
    IpoCycle := 4000,
    PosMode := 0,
    EndPos := EndPosition,
    VelocityMode := 3,
    Velocity := 5,
    Acceleration := 10,
    Deceleration := 10,
    Jerk := 50); // LS_2AxisLine

// NETWORK 11: ......
// NetworkDefaultComment
LS_2AxisLine_1(
    Axis0 := XAXIS,
    Axis1 := yAxis,
    Exec := LS_2AxisLine_0.Done,
    IpoCycle := 4000,
    PosMode := 0,
    EndPos := EndPosition1,
    VelocityMode := 3,
    Velocity := 5,
    Acceleration := 10,
    Deceleration := 10,
    Jerk := 50); // LS_2AxisLine
END_ACTION

END_PROGRAM

// Device/Application/POU_1
PROGRAM POU_1
VAR
    state        : INT := 0;
    
    mcPowerX     : MC_Power;
    mcPowerY     : MC_Power;
    
    mcMoveX_Fwd  : MC_MoveAbsolute;
    mcMoveX_Bck  : MC_MoveAbsolute;
    mcMoveY_Fwd  : MC_MoveAbsolute;
    mcMoveY_Bck  : MC_MoveAbsolute;
    
    mcRstX       : MC_Reset;
    mcRstY       : MC_Reset;
    resetX_exec  : BOOL := FALSE;
    resetY_exec  : BOOL := FALSE;
    
    start_test   : BOOL := FALSE;
    test_done    : BOOL := FALSE;
    error_flag   : BOOL := FALSE;
    error_id     : WORD;
END_VAR


(* ── Power ── *)
mcPowerX(Axis := XAXIS, Enable := TRUE, bRegulatorOn := TRUE, bDriveStart := TRUE);
mcPowerY(Axis := yAxis,  Enable := TRUE, bRegulatorOn := TRUE, bDriveStart := TRUE);

(* ── Reset blocks always called every scan ── *)
mcRstX(Axis := XAXIS, Execute := resetX_exec);
mcRstY(Axis := yAxis,  Execute := resetY_exec);

(* ── Move blocks ── *)
mcMoveX_Fwd(
    Axis         := XAXIS,
    Execute      := (state = 10),
    Position     := 1000.0,
    Velocity     := 1500.0,
    Acceleration := 2500.0,
    Deceleration := 2500.0,
    Jerk         := 5000.0,
    BufferMode   := 0
);

mcMoveX_Bck(
    Axis         := XAXIS,
    Execute      := (state = 20),
    Position     := 0.0,
    Velocity     := 300.0,
    Acceleration := 500.0,
    Deceleration := 500.0,
    Jerk         := 1500.0,
    BufferMode   := 0
);

mcMoveY_Fwd(
    Axis         := yAxis,
    Execute      := (state = 30),
    Position     := 500.0,
    Velocity     := 300.0,
    Acceleration := 500.0,
    Deceleration := 500.0,
    Jerk         := 1500.0,
    BufferMode   := 0
);

mcMoveY_Bck(
    Axis         := yAxis,
    Execute      := (state = 40),
    Position     := 0.0,
    Velocity     := 300.0,
    Acceleration := 500.0,
    Deceleration := 500.0,
    Jerk         := 1500.0,
    BufferMode   := 0
);

(* ── State Machine ── *)
CASE state OF

    0:
        test_done   := FALSE;
        error_flag  := FALSE;
        IF start_test AND mcPowerX.Status AND mcPowerY.Status THEN
            start_test := FALSE;
            state := 10;
        END_IF

    10: (* X forward to 1000mm *)
        IF mcMoveX_Fwd.Done THEN
            state := 20;
        ELSIF mcMoveX_Fwd.Error THEN
            error_id := mcMoveX_Fwd.ErrorID;
            state := 99;
        END_IF

    20: (* X return to 0 *)
        IF mcMoveX_Bck.Done THEN
            state := 30;
        ELSIF mcMoveX_Bck.Error THEN
            error_id := mcMoveX_Bck.ErrorID;
            state := 99;
        END_IF

    30: (* Y forward to 500mm *)
        IF mcMoveY_Fwd.Done THEN
            state := 40;
        ELSIF mcMoveY_Fwd.Error THEN
            error_id := mcMoveY_Fwd.ErrorID;
            state := 99;
        END_IF

    40: (* Y return to 0 *)
        IF mcMoveY_Bck.Done THEN
            test_done := TRUE;
            state := 0;
        ELSIF mcMoveY_Bck.Error THEN
            error_id := mcMoveY_Bck.ErrorID;
            state := 99;
        END_IF

    99: (* Error *)
        error_flag  := TRUE;
        resetX_exec := TRUE;
        resetY_exec := TRUE;
        IF mcRstX.Done AND mcRstY.Done THEN
            resetX_exec := FALSE;
            resetY_exec := FALSE;
            state := 0;
        END_IF

END_CASE

END_PROGRAM

// Device/Application/POU_3
PROGRAM POU_3
VAR
	test_output AT %QX1.4 : BOOL ;
END_VAR

test_output := TRUE;

END_PROGRAM
